FUNCTION_BLOCK DecimationDecorator IMPLEMENTS ITF_Analogue
VAR_INPUT
END_VAR
VAR_OUTPUT
END_VAR
VAR
END_VAR

{warning 'add method implementation '}
METHOD GetValue : INT
END_METHOD

END_FUNCTION_BLOCK

(* stored: Version 1.1.0.1, ProductVersion 3.1.4024.12
   POU DecimationDecorator: Id {489ffb12-88d5-4f8c-ae82-30974d4d0db9}, SpecialFunc None
   Method GetValue: Id {9e1632c3-3dab-40f9-9618-0a90b7bbe427} *)
